ABB RobotStudio station: practica4_20220517-120822.rsstn

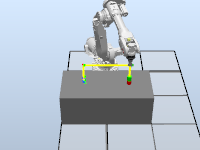
Station practica4 (saved by RobotStudio 20.4.9280.0)
Controller Controlador5
  mechanical unit ROB_1: IRB6640_180_255__04, 6 joints, base frame (0, 0, 0) mm
Layout (positions relative to the parent item):
  - Ventosa [mechanism] at (1500, 500, 1450) mm, rotated rx -180 ry 0 rz -180 deg
      TCP Ventosa at (0, 0, 200) mm
      links: PiezaVentosa
  - IRB6640_180_255__04 [mechanism, from Robots\IRB6640_180_255_G_04.rslib] at (0, 0, 0) mm; joint values [0.3218, 0.1103, 0.2349, 0, 1.2255, 0.3218] (rad or m)
  - Pieza_5 [part]
  - Pieza_6 [part]
  - Componente inteligente_1 [smart component]
      signals: DO PiezaDetectada, DO PiezaCogida, DI ActivaVentosa
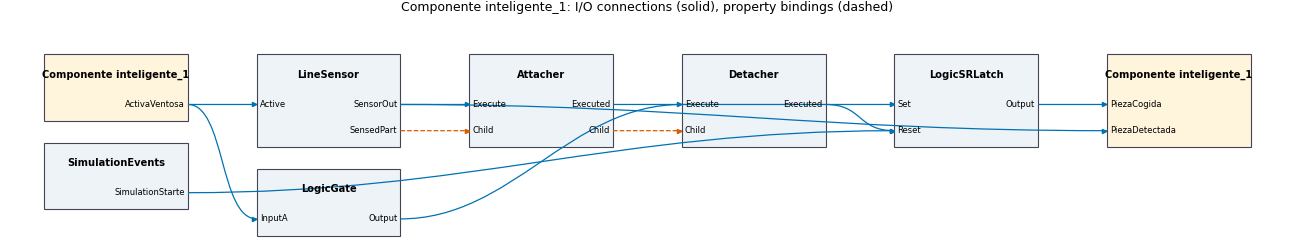
      connections:
        Componente inteligente_1.ActivaVentosa -> LineSensor.Active
        LineSensor.SensorOut -> Attacher.Execute
        Attacher.Executed -> LogicSRLatch.Set
        LogicSRLatch.Output -> Componente inteligente_1.PiezaCogida
        Componente inteligente_1.ActivaVentosa -> LogicGate.InputA
        LogicGate.Output -> Detacher.Execute
        Detacher.Executed -> LogicSRLatch.Reset
        SimulationEvents.SimulationStarted -> LogicSRLatch.Reset
        LineSensor.SensorOut -> Componente inteligente_1.PiezaDetectada
        LineSensor.SensedPart => Attacher.Child
        Attacher.Child => Detacher.Child
    - LineSensor [smart component, from Components\LineSensor.rslib] at (1500, 500, 1250) mm, rotated rx -180 ry 0 rz -180 deg
        properties: Start=[0 0 -0.002]; End=[0 0 0.02]; Radius=0.002; SensedPart=Pieza_8; SensedPoint=[1.5 0.5 0.95]
      - _sensorPart_ [part]
    - LogicSRLatch [smart component, from Components\LogicSRLatch.rslib]
    - SimulationEvents [smart component, from Components\SimulationEvents.rslib]
    - Attacher [smart component, from Components\Attacher.rslib]
        properties: Parent=Ventosa; Flange=0; Child=Pieza_8; Mount=false; Offset=[0 0 0]; Orientation=[0 0 0]
    - Detacher [smart component, from Components\Detacher.rslib]
        properties: Child=Pieza_8; KeepPosition=true
    - LogicGate [smart component, from Components\LogicGate.rslib]
        properties: Operator=NOT; Delay=0
  - Pieza_7 [part] at (0, 0, 0) mm
  - Pieza_8 [part] at (0, 0, 0) mm
Attachment: Ventosa is attached to IRB6640_180_255__04 / Link6
Attachment: LineSensor is attached to Ventosa / PiezaVentosa
Station logic (signal -> signal, property => property):
  Componente inteligente_1.PiezaDetectada -> Controlador5.ED_PiezaDetectada
  Controlador5.SD_ActivarVentosa -> Componente inteligente_1.ActivaVentosa
  Componente inteligente_1.PiezaCogida -> Controlador5.ED_PiezaCogida
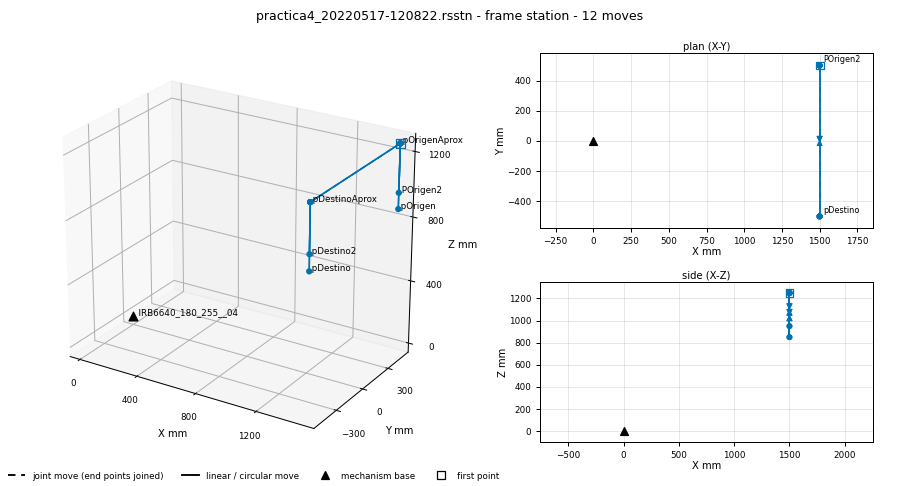
[picture p0: tool path of practica4_20220517-120822.rsstn in frame station, 12 of 12 moves have a stored position in this frame; points joined in program order, loops and branches not executed]
Targets, tools, work objects and paths stored in the station, written as RAPID:
! task T_ROB1
MODULE CalibData
  PERS tooldata Ventosa:=[TRUE,[[0,0,200],[1,0,0,0]],[1,[0,0,125],[1,0,0,0],0.002,0.002,0.001]];
ENDMODULE

! task T_ROB1
MODULE Module1
  CONST robtarget pOrigenBase:=[[1500,500,750],[0,0,1,0],[0,0,0,0],[9E+09,9E+09,9E+09,9E+09,9E+09,9E+09]];
  CONST robtarget pDestinoBase:=[[1500,-500,750],[0,0,1,0],[0,0,0,0],[9E+09,9E+09,9E+09,9E+09,9E+09,9E+09]];
  CONST robtarget pOrigen:=[[1500,500,850],[0,0,1,0],[0,0,0,0],[9E+09,9E+09,9E+09,9E+09,9E+09,9E+09]];
  CONST robtarget pDestino:=[[1500,-500,850],[0,0,1,0],[-1,0,-1,0],[9E+09,9E+09,9E+09,9E+09,9E+09,9E+09]];
  CONST robtarget pOrigenAprox:=[[1499.999958379,499.999981236,1249.999954428],[0.000000004,0,1,0.000000001],[0,-1,0,0],[9E+09,9E+09,9E+09,9E+09,9E+09,9E+09]];
  CONST robtarget pDestinoAprox:=[[1500,-500,1250],[0,0,1,0],[-1,0,-1,0],[9E+09,9E+09,9E+09,9E+09,9E+09,9E+09]];
  CONST robtarget POrigen2:=[[1500,500,950],[0,0,1,0],[0,0,0,0],[9E+09,9E+09,9E+09,9E+09,9E+09,9E+09]];
  CONST robtarget pDestino2:=[[1500,-500,950],[0,0,1,0],[-1,0,-1,0],[9E+09,9E+09,9E+09,9E+09,9E+09,9E+09]];
  PROC Path_10()
    MoveJ pOrigenAprox,v2500,z100,Ventosa\WObj:=wobj0;
    MoveL POrigen2,v1000,z100,Ventosa\WObj:=wobj0;
    MoveL pOrigenAprox,v300,z100,Ventosa\WObj:=wobj0;
    MoveJ pDestinoAprox,v2500,z100,Ventosa\WObj:=wobj0;
    MoveL pDestino,v300,fine,Ventosa\WObj:=wobj0;
    MoveL pDestinoAprox,v300,z100,Ventosa\WObj:=wobj0;
    MoveL pOrigenAprox,v1000,z100,Ventosa\WObj:=wobj0;
    MoveL pOrigen,v1000,z100,Ventosa\WObj:=wobj0;
    MoveL pOrigenAprox,v1000,z100,Ventosa\WObj:=wobj0;
    MoveL pDestinoAprox,v1000,z100,Ventosa\WObj:=wobj0;
    MoveL pDestino2,v1000,z100,Ventosa\WObj:=wobj0;
    MoveL pDestinoAprox,v1000,z100,Ventosa\WObj:=wobj0;
  ENDPROC
ENDMODULE

